(* IEC 61131-3 sources: com.logicals.lc3.webinar/logicals_Lib_Webinar/logicals_Webinar_Basic_Lib/logicals_Lib/src_C_Read_Localtime, 1 file *)

(* ---- logicals_Read_Localtime_C.iecst ---- *)
/*
 * ACHTUNG: Funktioniert NUR auf dem Raspberry Pi
 * Um auch die Uhrzeit in der Build-In-OLC lesen zu koennen MUSS die Funktion GetTime_C verwendet werden.
 */
{CustomImplementation}

NAMESPACE com.logicals.Basic.DateTime

FUNCTION FUN_lc_Read_Localtime_C
{ ImplementationProperties(functionHasCFile;) }

VAR_OUTPUT
    sec : DINT;
    min : DINT;
    hour : DINT;
    mday : DINT;
    mon : DINT;
    year : DINT;
    wday : DINT;
    yday : DINT;
    isdst : BOOL;
END_VAR

END_FUNCTION

END_NAMESPACE
